Staubli VAL3: clear.pgx

public program clear(num x_nX, num x_nY)
  local num i
  local num lLen
begin
  //-----------------------------------------------------------------------
  //Header begin
  //Description of program
  //  Erase the pY line from the column pX of the userPage.
  //
  //Input parameters
  //  num x_nX :
  //    role : Cursor column
  //    possible value : 0 to 39
  //  num x_nY :
  //    role : Cursor row
  //    possible value : 0 to 13
  //
  //Example
  //  call clear(15,8)
  //
  //History
  //  Creation : 28-04-08 - f.Rob
  //Header end
  //-----------------------------------------------------------------------
  call typeLen(x_nX,x_nY," ",40-x_nX)
  gotoxy(x_nX,x_nY)
end
